// SIMATIC S7-200 project (STEP 7-Micro/WIN), CPU 224 REL 02.01

ORGANIZATION_BLOCK PRINCIPAL:OB1
TITLE=COMENTARIOS DEL PROGRAMA
BEGIN
Network 1 // Título de segmento
// Comentario de segmento
LD     I0.0
LD     I0.1
O      M0.0
ALD
AN     M0.1
=      M0.0
Network 2
LD     I0.0
LD     I0.2
O      M0.1
ALD
AN     M0.0
=      M0.1
Network 3
LD     I0.3
EU
S      Q0.3, 2
Network 4
LD     I0.4
ED
R      Q0.3, 2
Network 5
LD     I0.0
A      I0.1
LD     I0.0
A      I0.2
OLD
AN     T40
=      M0.2
Network 6
LD     M0.2
TON    T40, +10
Network 7
LDW>=  T40, +5
=      Q0.6
Network 8
LD     Q0.6
LD     Q0.3
CTD    C20, +15
Network 9
LDN    C20
=      Q0.7
END_ORGANIZATION_BLOCK
